{attribute addProperty BoxType "EPP3744-0041-0016"}
{attribute addProperty Id "OutputAT %Q*ARRAY[0 ..1] OF BOOL1620"}
{attribute addProperty CRC "2653890939"}
{attribute addProperty SizeInBites "16"}
{attribute addProperty SizeInBytes "2"}
TYPE DIG_Outputs_0221D8A3 :
STRUCT
	{attribute addProperty Name "Output"}
	Output AT %Q* : ARRAY[0 ..1] OF BOOL;
END_STRUCT
END_TYPE

(* stored: Version 1.2.0.0, ProductVersion 3.1.4024.9
   DUT DIG_Outputs_0221D8A3: Id {523acf92-8c5b-43b9-9a71-8ce3931dac15} *)
